// TIA Portal V17 export
// export: Created 2024-09-02T12:50:08.3817091Z, ExportSetting WithDefaults, DisplayName Totally Integrated Automation Portal, DisplayVersion V17, DisplayName TIA Portal Openness, DisplayVersion V17, DisplayName TIA Portal Version Control Interface, DisplayVersion V17, DisplayName STEP 7 Professional, DisplayVersion V17, DisplayName STEP 7 Safety, DisplayVersion V17, DisplayName WinCC Professional, DisplayVersion V17
FUNCTION_BLOCK "GraFB1_FG02_Transport_OP70"   // FB1381, GRAPH
VERSION : 0.1
// stored: AcknowledgeErrorsRequired false, AutoNumber false, GraphVersion 4.0, InitialValuesAcquisition true, IsIECCheckEnabled false, LanguageInNetworks LAD, LockOperatingMode false, PermanentILProcessingInMANMode true, SetENOAutomatically false, SkipSteps false, UDAEnableTagReadback false, WithAlarmHandling true
   // inherited from GRAPH_BASE
   VAR
      OFF_SQ_BASE : Bool;
   END_VAR
   VAR_INPUT
      OFF_SQ { ExternalWritable := 'False'} : Bool := false;   // Kette ausschalten
      INIT_SQ { ExternalWritable := 'False'} : Bool := false;   // Kette in Initialzustand versetzen
      ACK_EF { ExternalWritable := 'False'} : Bool := false;   // Alle Fehler und Störungen quittieren
      S_PREV { ExternalWritable := 'False'} : Bool := false;   // Vorherigen Schritt am Parameter S_NO ausgeben
      S_NEXT { ExternalWritable := 'False'} : Bool := false;   // Nächsten Schritt am Parameter S_NO anzeigen
      SW_AUTO { ExternalWritable := 'False'} : Bool := false;   // Automtischer Betrieb
      SW_TAP { ExternalWritable := 'False'} : Bool := false;   // Halbautomatisch/Weiterschalten mit Transition
      SW_TOP { ExternalWritable := 'False'} : Bool := false;   // Halbautomatisch/Ignoriere Transition
      SW_MAN { ExternalWritable := 'False'} : Bool := false;   // Handbetrieb
      S_SEL { ExternalWritable := 'False'} : Int := 0;   // Schritt auswählen, der an S_NO ausgegeben werden soll
      S_ON { ExternalWritable := 'False'} : Bool := false;   // Schritt aktivieren, der an Parameter S_NO anliegt
      S_OFF { ExternalWritable := 'False'} : Bool := false;   // Schritt deaktivieren, der an Parameter S_NO anliegt
      T_PUSH { ExternalWritable := 'False'} : Bool := false;   // Schaltfreigabe für Transition im halbautomatischen Betrieb
   END_VAR
   VAR_OUTPUT
      S_NO { ExternalWritable := 'False'} : Int := 0;   // Schrittnummer
      S_MORE { ExternalWritable := 'False'} : Bool := false;   // Weitere Schritte sind vorhanden und können in S_NO angezeigt werden.
      S_ACTIVE { ExternalWritable := 'False'} : Bool := false;   // Schritt, der an Parameter S_NO angezeigt wird, ist aktiv
      ERR_FLT { ExternalWritable := 'False'} : Bool := false;   // Sammelfehler Interlock oder Supervision
      AUTO_ON { ExternalWritable := 'False'} : Bool := false;   // Automatischer Betrieb eingeschaltet
      TAP_ON { ExternalWritable := 'False'} : Bool := false;   // Halbautomatischer Betrieb/Schritt mit Transition eingeschaltet
      TOP_ON { ExternalWritable := 'False'} : Bool := false;   // Halbautomatischer Betrieb/Ignoriere Transition eingeschaltet
      MAN_ON { ExternalWritable := 'False'} : Bool := false;   // Handbetrieb eingeschaltet
   END_VAR
   VAR
      extBlock { S7_SetPoint := 'True'} : "LTLL_ManualGraphExt";
   END_VAR
BEGIN
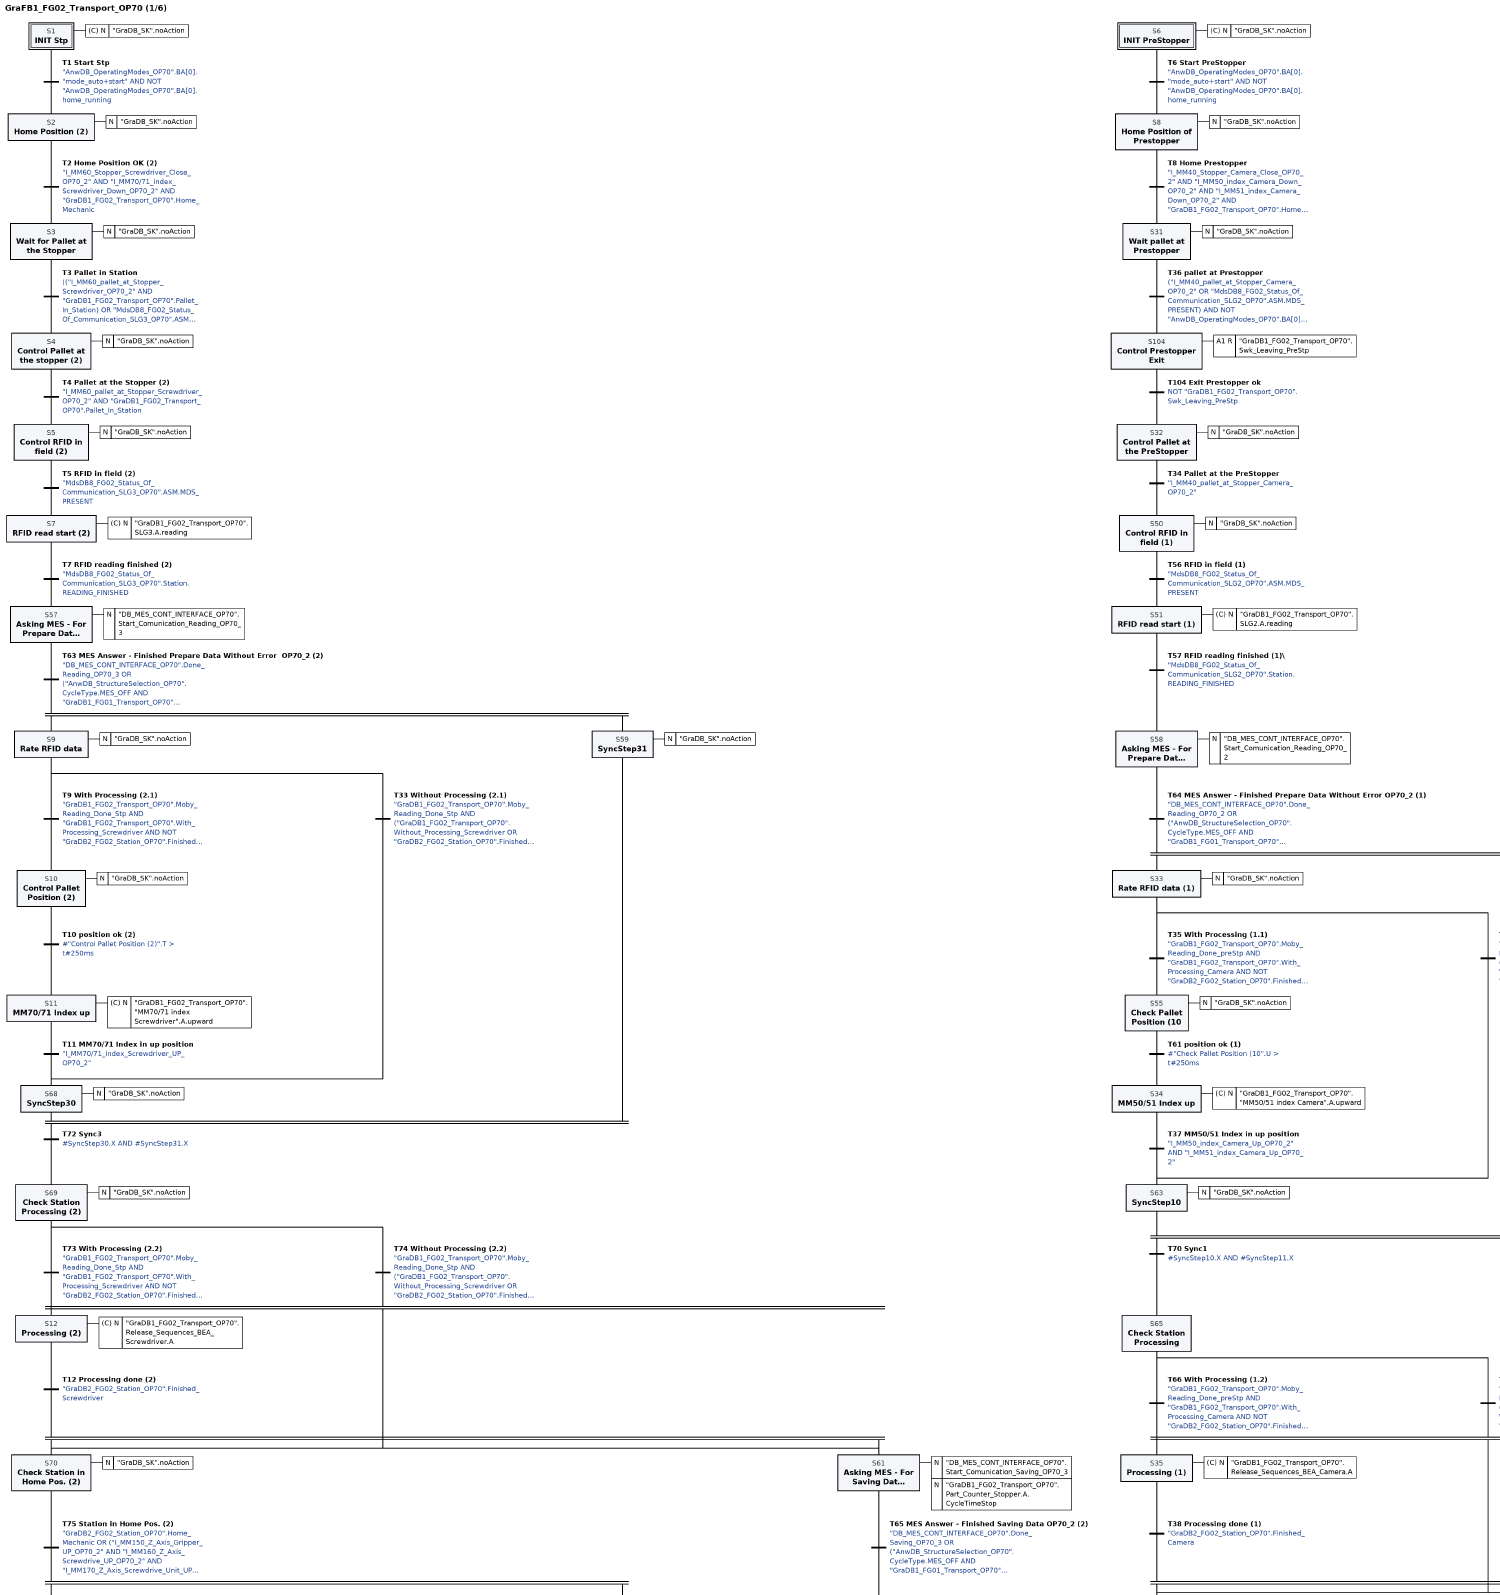
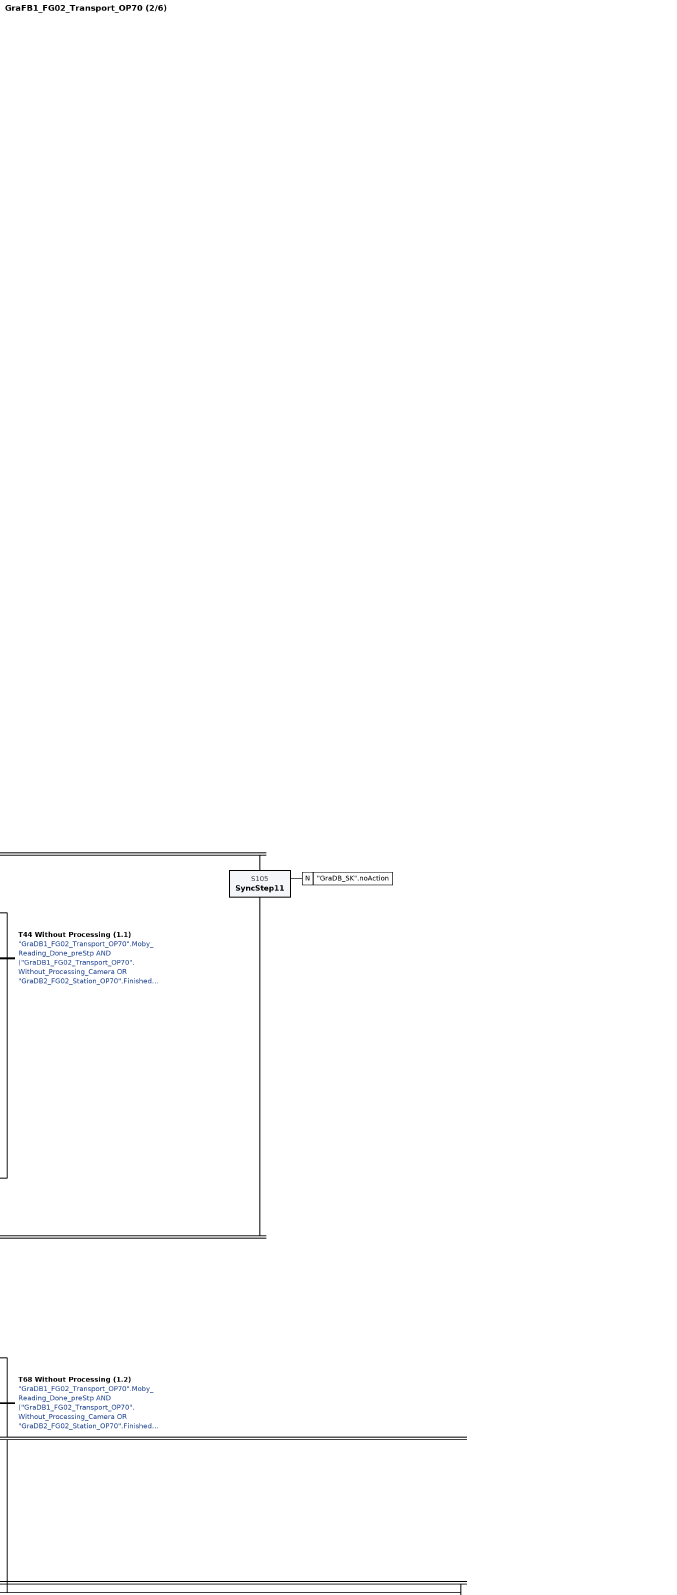
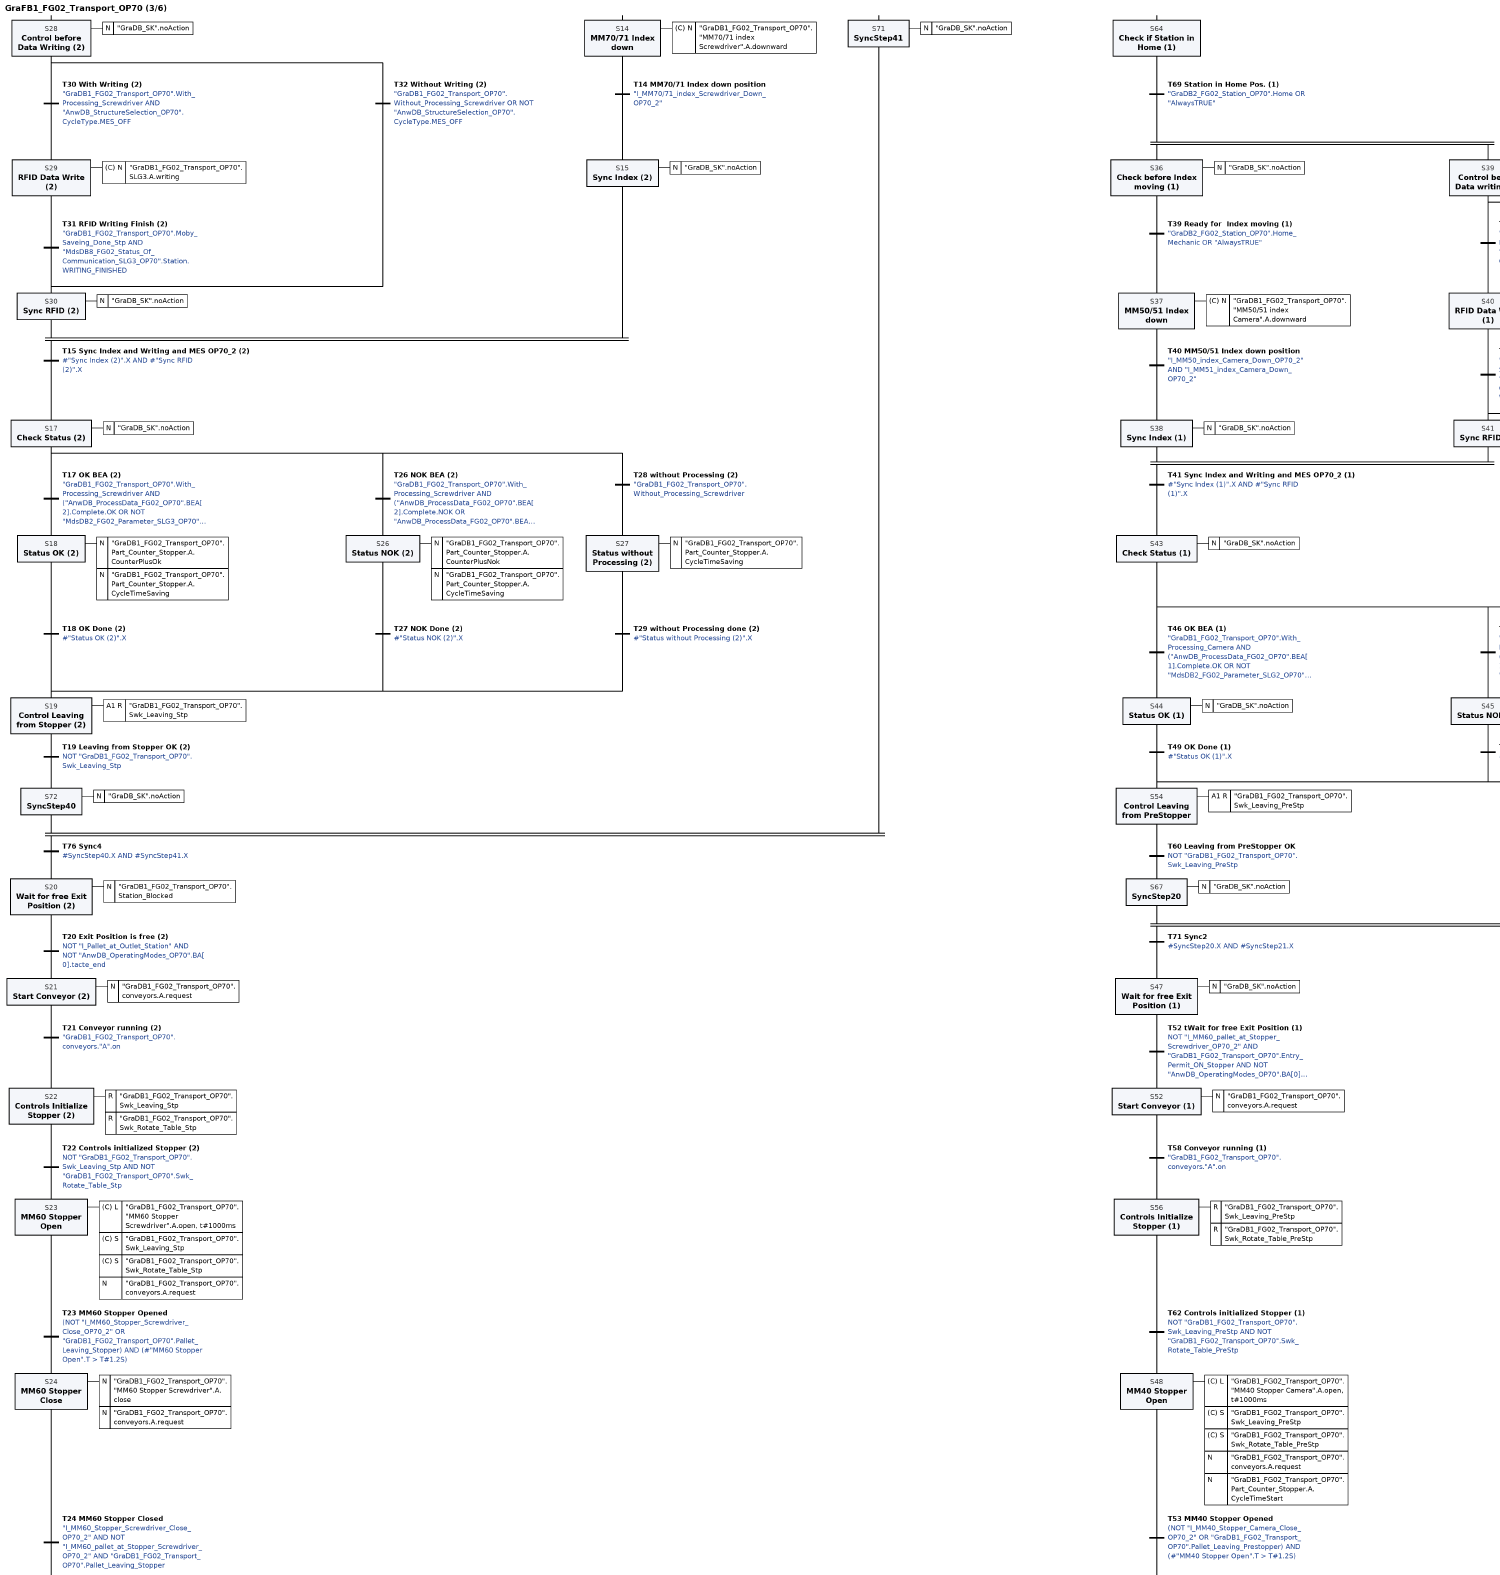
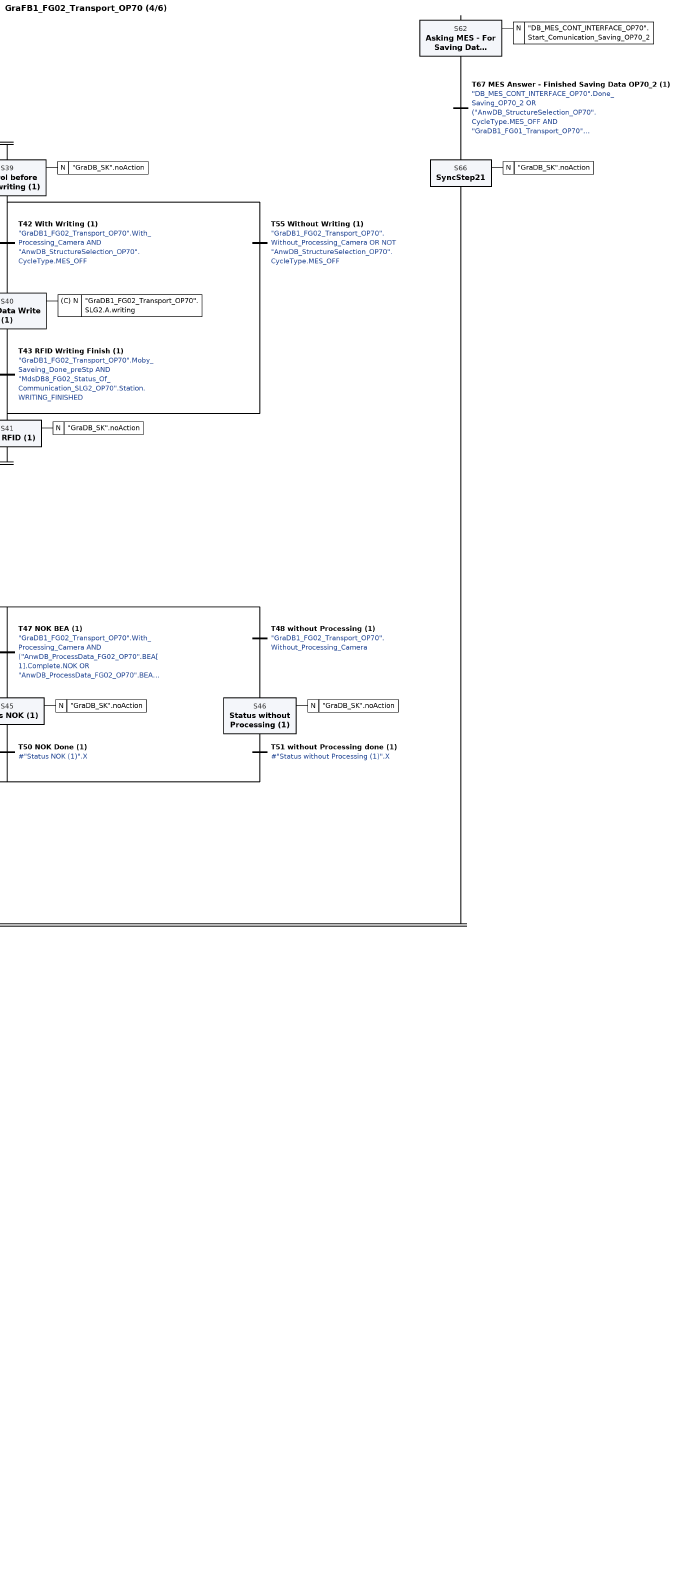
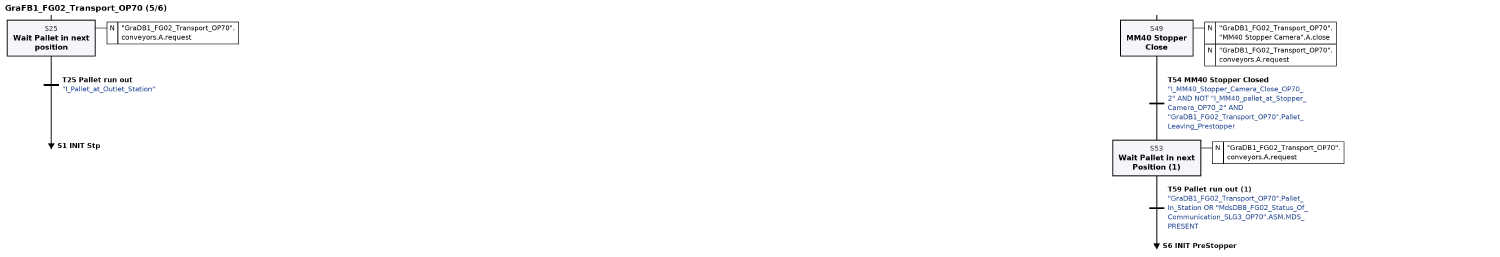
   // permanent pre-instructions
   NETWORK 1
   TITLE = HMI Lite Pass on data / HMI Lite Daten weiterreichen
      #extBlock.input := "LTLL_ManualGraphControl_OP70".screen[0].input;
   NETWORK 2
   TITLE = Instance DB Name query and pass on / Instanz DB Name abfragen und weiterreichen
      GetInstanceName(size := 0, OUT => #extBlock.input.instanceName);
   NETWORK 3
   TITLE = SK Mode
      "SysFC_SQ_Mode"(iFKT := 0, iTmsHalt := false, ioMOP := #RT_DATA.MOP);
   NETWORK 4
   TITLE = Signal change between pre-stopper and stopper / Signalwechsel Vorstopper/Stopper
      IF "GraDB1_FG02_Transport_OP70".Pallet_In_Station THEN
          "GraDB1_FG02_Transport_OP70".Swk_Leaving_PreStp := FALSE;
      END_IF;
      IF "I_Pallet_at_Outlet_Station" OR (NOT "GraDB1_FG02_Transport_OP70".Pallet_In_Station AND NOT "MdsDB8_FG02_Status_Of_Communication_SLG3_OP70".ASM.MDS_PRESENT AND NOT "I_MM60_pallet_at_Stopper_Screwdriver_OP70_2" AND "AlwaysFALSE") THEN
          "GraDB1_FG02_Transport_OP70".Swk_Leaving_Stp := FALSE;
      END_IF;
      IF "AlwaysTRUE" THEN "GraDB1_FG02_Transport_OP70".Swk_Rotate_Table_Stp := FALSE; END_IF;

   // sequencer 1: FG02 - Stopper MM60 / FG01 - Stopper
   INITIAL_STEP "INIT Stp":   // S1, max time T#10S, warning time T#7S
      interlock C := (none);   // Initialschritt / initial step
      supervision V := (none);   // Initialschritt / initial step
      (C)     N    "GraDB_SK".noAction
   END_STEP
   TRANSITION "Start Stp" FROM "INIT Stp" TO "Home Position (2)"   // T1
      := "AnwDB_OperatingModes_OP70".BA[0]."mode_auto+start" AND NOT "AnwDB_OperatingModes_OP70".BA[0].home_running;
   END_TRANSITION
   STEP "Home Position (2)":   // S2, max time T#10S, warning time T#7S
      supervision V := NOT #"Home Position OK (2)".TT AND (#"Home Position (2)".U > T#1S);
              N    "GraDB_SK".noAction
   END_STEP
   TRANSITION "Home Position OK (2)" FROM "Home Position (2)" TO "Wait for Pallet at the Stopper"   // T2
      := "I_MM60_Stopper_Screwdriver_Close_OP70_2" AND "I_MM70/71_index_Screwdriver_Down_OP70_2" AND "GraDB1_FG02_Transport_OP70".Home_Mechanic;
   END_TRANSITION
   STEP "Wait for Pallet at the Stopper":   // S3, max time T#10S, warning time T#7S
              N    "GraDB_SK".noAction
   END_STEP
   TRANSITION "Pallet in Station" FROM "Wait for Pallet at the Stopper" TO "Control Pallet at the stopper (2)"   // T3
      := (("I_MM60_pallet_at_Stopper_Screwdriver_OP70_2" AND "GraDB1_FG02_Transport_OP70".Pallet_In_Station) OR "MdsDB8_FG02_Status_Of_Communication_SLG3_OP70".ASM.MDS_PRESENT) AND NOT "AnwDB_OperatingModes_OP70".BA[0].tacte_end;
   END_TRANSITION
   STEP "Control Pallet at the stopper (2)":   // S4, max time T#10S, warning time T#7S
      supervision V := NOT #"Pallet at the Stopper (2)".TT AND (#"Control Pallet at the stopper (2)".U > T#5000mS);
              N    "GraDB_SK".noAction
   END_STEP
   TRANSITION "Pallet at the Stopper (2)" FROM "Control Pallet at the stopper (2)" TO "Control RFID in field (2)"   // T4
      := "I_MM60_pallet_at_Stopper_Screwdriver_OP70_2" AND "GraDB1_FG02_Transport_OP70".Pallet_In_Station;
   END_TRANSITION
   STEP "Rate RFID data":   // S9, max time T#10S, warning time T#7S
      interlock C := "MdsDB8_FG02_Status_Of_Communication_SLG3_OP70".Station.READING_FINISHED;
      supervision V := NOT #"With Processing (2.1)".TT AND NOT #"Without Processing (2.1)".TT AND (#"Rate RFID data".U > T#5000mS);
              N    "GraDB_SK".noAction
   END_STEP
   TRANSITION "With Processing (2.1)" FROM "Rate RFID data" TO "Control Pallet Position (2)"   // T9
      := "GraDB1_FG02_Transport_OP70".Moby_Reading_Done_Stp AND "GraDB1_FG02_Transport_OP70".With_Processing_Screwdriver AND NOT "GraDB2_FG02_Station_OP70".Finished_Screwdriver;
   END_TRANSITION
   TRANSITION "Without Processing (2.1)" FROM "Rate RFID data" TO SyncStep30   // T33
      := "GraDB1_FG02_Transport_OP70".Moby_Reading_Done_Stp AND ("GraDB1_FG02_Transport_OP70".Without_Processing_Screwdriver OR "GraDB2_FG02_Station_OP70".Finished_Screwdriver) AND (#"Rate RFID data".T > T#500MS);
   END_TRANSITION
   STEP "MM70/71 Index up":   // S11, max time T#10S, warning time T#7S
      interlock C := "I_MM150_Z_Axis_Gripper_UP_OP70_2" AND "I_MM160_Z_Axis_Screwdrive_UP_OP70_2" AND "I_MM170_Z_Axis_Screwdrive_Unit_UP_OP70_2";
      supervision V := NOT #"MM70/71 Index in up position".TT AND (#"MM70/71 Index up".U > T#5000mS);
      (C)     N    "GraDB1_FG02_Transport_OP70"."MM70/71 index Screwdriver".A.upward
   END_STEP
   TRANSITION "MM70/71 Index in up position" FROM "MM70/71 Index up" TO SyncStep30   // T11
      := "I_MM70/71_index_Screwdriver_UP_OP70_2";
   END_TRANSITION
   STEP "Processing (2)":   // S12, max time T#10S, warning time T#7S
      interlock C := "MdsDB8_FG02_Status_Of_Communication_SLG3_OP70".Station.READING_FINISHED;
      (C)     N    "GraDB1_FG02_Transport_OP70".Release_Sequences_BEA_Screwdriver.A
   END_STEP
   TRANSITION "Processing done (2)" FROM "Processing (2)" TO ("Check Station in Home Pos. (2)", "Asking MES - For Saving Data OP70_2 (2)")   // T12
      := "GraDB2_FG02_Station_OP70".Finished_Screwdriver;
   END_TRANSITION
   STEP "MM70/71 Index  down":   // S14, max time T#10S, warning time T#7S
      interlock C := "I_MM150_Z_Axis_Gripper_UP_OP70_2" AND "I_MM160_Z_Axis_Screwdrive_UP_OP70_2" AND "I_MM170_Z_Axis_Screwdrive_Unit_UP_OP70_2";
      supervision V := NOT #"MM70/71 Index down position".TT AND (#"MM70/71 Index  down".U > T#5s);
      (C)     N    "GraDB1_FG02_Transport_OP70"."MM70/71 index Screwdriver".A.downward
   END_STEP
   TRANSITION "MM70/71 Index down position" FROM "MM70/71 Index  down" TO "Sync Index (2)"   // T14
      := "I_MM70/71_index_Screwdriver_Down_OP70_2";
   END_TRANSITION
   STEP "Sync Index (2)":   // S15, max time T#10S, warning time T#7S
              N    "GraDB_SK".noAction
   END_STEP
   STEP "Control before Data Writing (2)":   // S28, max time T#10S, warning time T#7S
              N    "GraDB_SK".noAction
   END_STEP
   TRANSITION "With Writing (2)" FROM "Control before Data Writing (2)" TO "RFID Data Write (2)"   // T30
      := "GraDB1_FG02_Transport_OP70".With_Processing_Screwdriver AND "AnwDB_StructureSelection_OP70".CycleType.MES_OFF;
   END_TRANSITION
   TRANSITION "Without Writing (2)" FROM "Control before Data Writing (2)" TO "Sync RFID (2)"   // T32
      := "GraDB1_FG02_Transport_OP70".Without_Processing_Screwdriver OR NOT "AnwDB_StructureSelection_OP70".CycleType.MES_OFF;
   END_TRANSITION
   STEP "RFID Data Write (2)":   // S29, max time T#10S, warning time T#7S
      interlock C := "GraDB1_FG02_Transport_OP70".Moby_Reading_Done_Stp;
      supervision V := NOT #"RFID Writing Finish (2)".TT AND (#"RFID Data Write (2)".U > T#5000MS);
      (C)     N    "GraDB1_FG02_Transport_OP70".SLG3.A.writing
   END_STEP
   TRANSITION "RFID Writing Finish (2)" FROM "RFID Data Write (2)" TO "Sync RFID (2)"   // T31
      := "GraDB1_FG02_Transport_OP70".Moby_Saveing_Done_Stp AND "MdsDB8_FG02_Status_Of_Communication_SLG3_OP70".Station.WRITING_FINISHED;
   END_TRANSITION
   STEP "Sync RFID (2)":   // S30, max time T#10S, warning time T#7S
              N    "GraDB_SK".noAction
   END_STEP
   TRANSITION "Sync Index and Writing and MES OP70_2 (2)" FROM ("Sync Index (2)", "Sync RFID (2)") TO "Check Status (2)"   // T15
      := #"Sync Index (2)".X AND #"Sync RFID (2)".X;
   END_TRANSITION
   STEP "Check Status (2)":   // S17, max time T#10S, warning time T#7S
      supervision V := NOT #"OK BEA (2)".TT AND NOT #"OK BEA (2)".TT AND NOT #"without Processing (2)".TT AND (#"Check Status (2)".U > T#1000MS);
              N    "GraDB_SK".noAction
   END_STEP
   TRANSITION "OK BEA (2)" FROM "Check Status (2)" TO "Status OK (2)"   // T17
      := "GraDB1_FG02_Transport_OP70".With_Processing_Screwdriver AND ("AnwDB_ProcessData_FG02_OP70".BEA[2].Complete.OK OR NOT "MdsDB2_FG02_Parameter_SLG3_OP70".Release_BEA[2]) AND ("AnwDB_ProcessData_FG02_OP70".BEA[3].Complete.OK OR NOT "MdsDB2_FG02_Parameter_SLG3_OP70".Release_BEA[3]);
   END_TRANSITION
   TRANSITION "NOK BEA (2)" FROM "Check Status (2)" TO "Status NOK (2)"   // T26
      := "GraDB1_FG02_Transport_OP70".With_Processing_Screwdriver AND ("AnwDB_ProcessData_FG02_OP70".BEA[2].Complete.NOK OR "AnwDB_ProcessData_FG02_OP70".BEA[2].Complete.NOK_Active OR "AnwDB_ProcessData_FG02_OP70".BEA[3].Complete.NOK OR "AnwDB_ProcessData_FG02_OP70".BEA[3].Complete.NOK_Active);
   END_TRANSITION
   TRANSITION "without Processing (2)" FROM "Check Status (2)" TO "Status without Processing (2)"   // T28
      := "GraDB1_FG02_Transport_OP70".Without_Processing_Screwdriver;
   END_TRANSITION
   STEP "Status OK (2)":   // S18, max time T#10S, warning time T#7S
              N    "GraDB1_FG02_Transport_OP70".Part_Counter_Stopper.A.CounterPlusOk
              N    "GraDB1_FG02_Transport_OP70".Part_Counter_Stopper.A.CycleTimeSaving
   END_STEP
   TRANSITION "OK Done (2)" FROM "Status OK (2)" TO "Control Leaving from Stopper (2)"   // T18
      := #"Status OK (2)".X;
   END_TRANSITION
   STEP "Status NOK (2)":   // S26, max time T#10S, warning time T#7S
              N    "GraDB1_FG02_Transport_OP70".Part_Counter_Stopper.A.CounterPlusNok
              N    "GraDB1_FG02_Transport_OP70".Part_Counter_Stopper.A.CycleTimeSaving
   END_STEP
   TRANSITION "NOK Done (2)" FROM "Status NOK (2)" TO "Control Leaving from Stopper (2)"   // T27
      := #"Status NOK (2)".X;
   END_TRANSITION
   STEP "Status without Processing (2)":   // S27, max time T#10S, warning time T#7S
              N    "GraDB1_FG02_Transport_OP70".Part_Counter_Stopper.A.CycleTimeSaving
   END_STEP
   TRANSITION "without Processing done (2)" FROM "Status without Processing (2)" TO "Control Leaving from Stopper (2)"   // T29
      := #"Status without Processing (2)".X;
   END_TRANSITION
   STEP "Wait for free Exit Position (2)":   // S20, max time T#10S, warning time T#7S
              N    "GraDB1_FG02_Transport_OP70".Station_Blocked
   END_STEP
   TRANSITION "Exit Position is free (2)" FROM "Wait for free Exit Position (2)" TO "Start Conveyor (2)"   // T20
      := NOT "I_Pallet_at_Outlet_Station" AND NOT "AnwDB_OperatingModes_OP70".BA[0].tacte_end;
   END_TRANSITION
   STEP "MM60 Stopper Open":   // S23, max time T#10S, warning time T#7S
      interlock C := NOT "I_Pallet_at_Outlet_Station";
      supervision V := NOT #"MM60 Stopper Opened".TT AND (#"MM60 Stopper Open".U > T#5000mS);
      (C)     L    "GraDB1_FG02_Transport_OP70"."MM60 Stopper Screwdriver".A.open, t#1000ms
      (C)     S    "GraDB1_FG02_Transport_OP70".Swk_Leaving_Stp
      (C)     S    "GraDB1_FG02_Transport_OP70".Swk_Rotate_Table_Stp
              N    "GraDB1_FG02_Transport_OP70".conveyors.A.request
   END_STEP
   TRANSITION "MM60 Stopper Opened" FROM "MM60 Stopper Open" TO "MM60 Stopper Close"   // T23
      := (NOT "I_MM60_Stopper_Screwdriver_Close_OP70_2" OR "GraDB1_FG02_Transport_OP70".Pallet_Leaving_Stopper) AND (#"MM60 Stopper Open".T > T#1.2S);
   END_TRANSITION
   STEP "MM60 Stopper Close":   // S24, max time T#10S, warning time T#7S
      supervision V := NOT #"MM60 Stopper Closed".TT AND (#"MM60 Stopper Close".U > T#5000mS);
              N    "GraDB1_FG02_Transport_OP70"."MM60 Stopper Screwdriver".A.close
              N    "GraDB1_FG02_Transport_OP70".conveyors.A.request
   END_STEP
   TRANSITION "MM60 Stopper Closed" FROM "MM60 Stopper Close" TO "Wait Pallet in next position"   // T24
      := "I_MM60_Stopper_Screwdriver_Close_OP70_2" AND NOT "I_MM60_pallet_at_Stopper_Screwdriver_OP70_2" AND "GraDB1_FG02_Transport_OP70".Pallet_Leaving_Stopper;
   END_TRANSITION
   STEP "Control RFID in field (2)":   // S5, max time T#10S, warning time T#7S
      supervision V := NOT #"RFID in field (2)".TT AND (#"Control RFID in field (2)".U > T#5000mS);
              N    "GraDB_SK".noAction
   END_STEP
   TRANSITION "RFID in field (2)" FROM "Control RFID in field (2)" TO "RFID read start (2)"   // T5
      := "MdsDB8_FG02_Status_Of_Communication_SLG3_OP70".ASM.MDS_PRESENT;
   END_TRANSITION
   STEP "RFID read start (2)":   // S7, max time T#10S, warning time T#7S
      interlock C := "MdsDB8_FG02_Status_Of_Communication_SLG3_OP70".ASM.MDS_PRESENT;
      supervision V := NOT #"RFID reading finished (2)".TT AND (#"RFID read start (2)".U > T#5000mS);
      (C)     N    "GraDB1_FG02_Transport_OP70".SLG3.A.reading
   END_STEP
   TRANSITION "RFID reading finished (2)" FROM "RFID read start (2)" TO "Asking MES - For Prepare Data  OP70_2 (2)"   // T7
      := "MdsDB8_FG02_Status_Of_Communication_SLG3_OP70".Station.READING_FINISHED;
   END_TRANSITION
   STEP "Start Conveyor (2)":   // S21, max time T#10S, warning time T#7S
      supervision V := NOT #"Conveyor running (2)".TT AND (#"Start Conveyor (2)".U > T#5000MS);
              N    "GraDB1_FG02_Transport_OP70".conveyors.A.request
   END_STEP
   TRANSITION "Conveyor running (2)" FROM "Start Conveyor (2)" TO "Controls Initialize Stopper (2)"   // T21
      := "GraDB1_FG02_Transport_OP70".conveyors."A".on;
   END_TRANSITION
   STEP "Wait Pallet in next position":   // S25, max time T#10S, warning time T#7S
      supervision V := NOT #"Pallet run out".TT AND (#"Wait Pallet in next position".U > T#25000MS);
              N    "GraDB1_FG02_Transport_OP70".conveyors.A.request
   END_STEP
   TRANSITION "Pallet run out" FROM "Wait Pallet in next position" TO "INIT Stp"   // T25, jump
      := "I_Pallet_at_Outlet_Station";
   END_TRANSITION
   STEP "Control Leaving from Stopper (2)":   // S19, max time T#10S, warning time T#7S
      supervision V := NOT #"Leaving from Stopper OK (2)".TT AND (#"Control Leaving from Stopper (2)".U > T#1000MS);
          A1  R    "GraDB1_FG02_Transport_OP70".Swk_Leaving_Stp
   END_STEP
   TRANSITION "Leaving from Stopper OK (2)" FROM "Control Leaving from Stopper (2)" TO SyncStep40   // T19
      := NOT "GraDB1_FG02_Transport_OP70".Swk_Leaving_Stp;
   END_TRANSITION
   STEP "Control Pallet Position (2)":   // S10, max time T#10S, warning time T#7S
      supervision V := NOT #"position ok (2)".TT AND (#"Control Pallet Position (2)".U > T#5000MS);
              N    "GraDB_SK".noAction
   END_STEP
   TRANSITION "position ok (2)" FROM "Control Pallet Position (2)" TO "MM70/71 Index up"   // T10
      := #"Control Pallet Position (2)".T > t#250ms;
   END_TRANSITION
   STEP "Controls Initialize Stopper (2)":   // S22, max time T#10S, warning time T#7S
      supervision V := NOT #"Controls initialized Stopper (2)".TT AND (#"Controls Initialize Stopper (2)".U > T#1000MS);
              R    "GraDB1_FG02_Transport_OP70".Swk_Leaving_Stp
              R    "GraDB1_FG02_Transport_OP70".Swk_Rotate_Table_Stp
   END_STEP
   TRANSITION "Controls initialized Stopper (2)" FROM "Controls Initialize Stopper (2)" TO "MM60 Stopper Open"   // T22
      := NOT "GraDB1_FG02_Transport_OP70".Swk_Leaving_Stp AND NOT "GraDB1_FG02_Transport_OP70".Swk_Rotate_Table_Stp;
   END_TRANSITION
   STEP SyncStep30:   // S68, max time T#10S, warning time T#7S
              N    "GraDB_SK".noAction
   END_STEP
   STEP SyncStep40:   // S72, max time T#10S, warning time T#7S
              N    "GraDB_SK".noAction
   END_STEP
   STEP SyncStep31:   // S59, max time T#10S, warning time T#7S
              N    "GraDB_SK".noAction
   END_STEP
   TRANSITION Sync3 FROM (SyncStep30, SyncStep31) TO "Check Station Processing (2)"   // T72
      := #SyncStep30.X AND #SyncStep31.X;
   END_TRANSITION
   STEP "Check Station Processing (2)":   // S69, max time T#10S, warning time T#7S
              N    "GraDB_SK".noAction
   END_STEP
   TRANSITION "With Processing (2.2)" FROM "Check Station Processing (2)" TO "Processing (2)"   // T73
      := "GraDB1_FG02_Transport_OP70".Moby_Reading_Done_Stp AND "GraDB1_FG02_Transport_OP70".With_Processing_Screwdriver AND NOT "GraDB2_FG02_Station_OP70".Finished_Screwdriver;
   END_TRANSITION
   TRANSITION "Without Processing (2.2)" FROM "Check Station Processing (2)" TO ("Check Station in Home Pos. (2)", "Asking MES - For Saving Data OP70_2 (2)")   // T74
      := "GraDB1_FG02_Transport_OP70".Moby_Reading_Done_Stp AND ("GraDB1_FG02_Transport_OP70".Without_Processing_Screwdriver OR "GraDB2_FG02_Station_OP70".Finished_Screwdriver) AND (#"Check Station Processing (2)".T > t#500ms);
   END_TRANSITION
   STEP "Check Station in Home Pos. (2)":   // S70, max time T#10S, warning time T#7S
      supervision V := NOT #"Station in Home Pos. (2)".TT AND (#"Check Station in Home Pos. (2)".U > T#5s);
              N    "GraDB_SK".noAction
   END_STEP
   TRANSITION "Station in Home Pos. (2)" FROM "Check Station in Home Pos. (2)" TO ("Control before Data Writing (2)", "MM70/71 Index  down")   // T75
      := "GraDB2_FG02_Station_OP70".Home_Mechanic OR ("I_MM150_Z_Axis_Gripper_UP_OP70_2" AND "I_MM160_Z_Axis_Screwdrive_UP_OP70_2" AND "I_MM170_Z_Axis_Screwdrive_Unit_UP_OP70_2");
   END_TRANSITION
   STEP SyncStep41:   // S71, max time T#10S, warning time T#7S
              N    "GraDB_SK".noAction
   END_STEP
   TRANSITION Sync4 FROM (SyncStep40, SyncStep41) TO "Wait for free Exit Position (2)"   // T76
      := #SyncStep40.X AND #SyncStep41.X;
   END_TRANSITION
   STEP "Asking MES - For Saving Data OP70_2 (2)":   // S61, max time T#10S, warning time T#7S
      interlock C := "MdsDB8_FG02_Status_Of_Communication_SLG3_OP70".ASM.MDS_PRESENT;
      supervision V := NOT #"MES Answer - Finished Saving Data OP70_2 (2)".TT AND (#"Asking MES - For Saving Data OP70_2 (2)".U > T#5000mS) AND "AlwaysFALSE";
              N    "DB_MES_CONT_INTERFACE_OP70".Start_Comunication_Saving_OP70_3
              N    "GraDB1_FG02_Transport_OP70".Part_Counter_Stopper.A.CycleTimeStop
   END_STEP
   TRANSITION "MES Answer - Finished Saving Data OP70_2 (2)" FROM "Asking MES - For Saving Data OP70_2 (2)" TO SyncStep41   // T65
      := "DB_MES_CONT_INTERFACE_OP70".Done_Saving_OP70_3 OR ("AnwDB_StructureSelection_OP70".CycleType.MES_OFF AND "GraDB1_FG01_Transport_OP70".Tracebility_off) OR "AnwDB_StructureSelection_OP70".UserDefine.IbmMode;
   END_TRANSITION
   STEP "Asking MES - For Prepare Data  OP70_2 (2)":   // S57, max time T#10S, warning time T#7S
      interlock C := "MdsDB8_FG02_Status_Of_Communication_SLG3_OP70".ASM.MDS_PRESENT;
      supervision V := NOT #"MES Answer - Finished Prepare Data Without Error  OP70_2 (2)".TT AND (#"Asking MES - For Prepare Data  OP70_2 (2)".U > T#7s);
              N    "DB_MES_CONT_INTERFACE_OP70".Start_Comunication_Reading_OP70_3
   END_STEP
   TRANSITION "MES Answer - Finished Prepare Data Without Error  OP70_2 (2)" FROM "Asking MES - For Prepare Data  OP70_2 (2)" TO ("Rate RFID data", SyncStep31)   // T63
      := "DB_MES_CONT_INTERFACE_OP70".Done_Reading_OP70_3 OR ("AnwDB_StructureSelection_OP70".CycleType.MES_OFF AND "GraDB1_FG01_Transport_OP70".Tracebility_off) OR "AnwDB_StructureSelection_OP70".UserDefine.IbmMode;
   END_TRANSITION

   // sequencer 2: FG02 - PreStopper MM40 / FG01 - Vorstopper
   INITIAL_STEP "INIT PreStopper":   // S6, max time T#10S, warning time T#7S
      interlock C := (none);   // Initialschritt / initial step
      supervision V := (none);   // Initialschritt / initial step
      (C)     N    "GraDB_SK".noAction
   END_STEP
   TRANSITION "Start PreStopper" FROM "INIT PreStopper" TO "Home Position of Prestopper"   // T6
      := "AnwDB_OperatingModes_OP70".BA[0]."mode_auto+start" AND NOT "AnwDB_OperatingModes_OP70".BA[0].home_running;
   END_TRANSITION
   STEP "Home Position of Prestopper":   // S8, max time T#10S, warning time T#7S
      supervision V := NOT #"Home Prestopper".TT AND (#"Home Position of Prestopper".U > T#1S);
              N    "GraDB_SK".noAction
   END_STEP
   TRANSITION "Home Prestopper" FROM "Home Position of Prestopper" TO "Wait pallet at Prestopper"   // T8
      := "I_MM40_Stopper_Camera_Close_OP70_2" AND "I_MM50_index_Camera_Down_OP70_2" AND "I_MM51_index_Camera_Down_OP70_2" AND "GraDB1_FG02_Transport_OP70".Home_Mechanic;
   END_TRANSITION
   STEP "Sync Index (1)":   // S38, max time T#10S, warning time T#7S
              N    "GraDB_SK".noAction
   END_STEP
   STEP "Control before Data writing (1)":   // S39, max time T#10S, warning time T#7S
              N    "GraDB_SK".noAction
   END_STEP
   TRANSITION "With Writing (1)" FROM "Control before Data writing (1)" TO "RFID Data Write (1)"   // T42
      := "GraDB1_FG02_Transport_OP70".With_Processing_Camera AND "AnwDB_StructureSelection_OP70".CycleType.MES_OFF;
   END_TRANSITION
   TRANSITION "Without Writing (1)" FROM "Control before Data writing (1)" TO "Sync RFID (1)"   // T55
      := "GraDB1_FG02_Transport_OP70".Without_Processing_Camera OR NOT "AnwDB_StructureSelection_OP70".CycleType.MES_OFF;
   END_TRANSITION
   STEP "Rate RFID data (1)":   // S33, max time T#10S, warning time T#7S
      interlock C := "AlwaysTRUE";
      supervision V := NOT #"With Processing (1.1)".TT AND NOT #"Without Processing (1.1)".TT AND (#"Rate RFID data (1)".U > T#5000mS);
              N    "GraDB_SK".noAction
   END_STEP
   TRANSITION "With Processing (1.1)" FROM "Rate RFID data (1)" TO "Check Pallet Position (10"   // T35
      := "GraDB1_FG02_Transport_OP70".Moby_Reading_Done_preStp AND "GraDB1_FG02_Transport_OP70".With_Processing_Camera AND NOT "GraDB2_FG02_Station_OP70".Finished_Camera;
   END_TRANSITION
   TRANSITION "Without Processing (1.1)" FROM "Rate RFID data (1)" TO SyncStep10   // T44
      := "GraDB1_FG02_Transport_OP70".Moby_Reading_Done_preStp AND ("GraDB1_FG02_Transport_OP70".Without_Processing_Camera OR "GraDB2_FG02_Station_OP70".Finished_Camera) AND (#"Rate RFID data (1)".T > T#500MS);
   END_TRANSITION
   STEP "Processing (1)":   // S35, max time T#10S, warning time T#7S
      interlock C := "I_MM50_index_Camera_Up_OP70_2" AND "I_MM51_index_Camera_Up_OP70_2" AND "MdsDB8_FG02_Status_Of_Communication_SLG2_OP70".Station.READING_FINISHED;
      (C)     N    "GraDB1_FG02_Transport_OP70".Release_Sequences_BEA_Camera.A
   END_STEP
   TRANSITION "Processing done (1)" FROM "Processing (1)" TO ("Check if Station in Home (1)", "Asking MES - For Saving Data OP70_2 (1)")   // T38
      := "GraDB2_FG02_Station_OP70".Finished_Camera;
   END_TRANSITION
   STEP "RFID Data Write (1)":   // S40, max time T#10S, warning time T#7S
      interlock C := "GraDB1_FG02_Transport_OP70".Moby_Reading_Done_preStp;
      supervision V := NOT #"RFID Writing Finish (1)".TT AND (#"RFID Data Write (1)".U > T#5000MS);
      (C)     N    "GraDB1_FG02_Transport_OP70".SLG2.A.writing
   END_STEP
   TRANSITION "RFID Writing Finish (1)" FROM "RFID Data Write (1)" TO "Sync RFID (1)"   // T43
      := "GraDB1_FG02_Transport_OP70".Moby_Saveing_Done_preStp AND "MdsDB8_FG02_Status_Of_Communication_SLG2_OP70".Station.WRITING_FINISHED;
   END_TRANSITION
   STEP "Check before Index moving (1)":   // S36, max time T#10S, warning time T#7S
      interlock C := "AlwaysTRUE";
      supervision V := NOT #"Ready for  Index moving (1)".TT AND (#"Check before Index moving (1)".U > T#5000MS);
              N    "GraDB_SK".noAction
   END_STEP
   TRANSITION "Ready for  Index moving (1)" FROM "Check before Index moving (1)" TO "MM50/51 Index  down"   // T39
      := "GraDB2_FG02_Station_OP70".Home_Mechanic OR "AlwaysTRUE";
   END_TRANSITION
   STEP "MM50/51 Index up":   // S34, max time T#10S, warning time T#7S
      supervision V := NOT #"MM50/51 Index in up position".TT AND (#"MM50/51 Index up".U > T#5000mS);
      (C)     N    "GraDB1_FG02_Transport_OP70"."MM50/51 index Camera".A.upward
   END_STEP
   TRANSITION "MM50/51 Index in up position" FROM "MM50/51 Index up" TO SyncStep10   // T37
      := "I_MM50_index_Camera_Up_OP70_2" AND "I_MM51_index_Camera_Up_OP70_2";
   END_TRANSITION
   STEP "MM50/51 Index  down":   // S37, max time T#10S, warning time T#7S
      interlock C := "AlwaysTRUE";
      supervision V := NOT #"MM50/51 Index down position".TT AND (#"MM50/51 Index  down".U > T#5000mS);
      (C)     N    "GraDB1_FG02_Transport_OP70"."MM50/51 index Camera".A.downward
   END_STEP
   TRANSITION "MM50/51 Index down position" FROM "MM50/51 Index  down" TO "Sync Index (1)"   // T40
      := "I_MM50_index_Camera_Down_OP70_2" AND "I_MM51_index_Camera_Down_OP70_2";
   END_TRANSITION
   STEP "Wait pallet at Prestopper":   // S31, max time T#10S, warning time T#7S
              N    "GraDB_SK".noAction
   END_STEP
   TRANSITION "pallet at Prestopper" FROM "Wait pallet at Prestopper" TO "Control Prestopper Exit"   // T36
      := ("I_MM40_pallet_at_Stopper_Camera_OP70_2" OR "MdsDB8_FG02_Status_Of_Communication_SLG2_OP70".ASM.MDS_PRESENT) AND NOT "AnwDB_OperatingModes_OP70".BA[0].tacte_end;
   END_TRANSITION
   STEP "Control Pallet at the PreStopper":   // S32, max time T#10S, warning time T#7S
      supervision V := NOT #"Pallet at the PreStopper".TT AND (#"Control Pallet at the PreStopper".U > T#5000mS);
              N    "GraDB_SK".noAction
   END_STEP
   TRANSITION "Pallet at the PreStopper" FROM "Control Pallet at the PreStopper" TO "Control RFID in field (1)"   // T34
      := "I_MM40_pallet_at_Stopper_Camera_OP70_2";
   END_TRANSITION
   STEP "Sync RFID (1)":   // S41, max time T#10S, warning time T#7S
              N    "GraDB_SK".noAction
   END_STEP
   TRANSITION "Sync Index and Writing and MES OP70_2 (1)" FROM ("Sync Index (1)", "Sync RFID (1)") TO "Check Status (1)"   // T41
      := #"Sync Index (1)".X AND #"Sync RFID (1)".X;
   END_TRANSITION
   STEP "Check Status (1)":   // S43, max time T#10S, warning time T#7S
      supervision V := NOT #"OK BEA (1)".TT AND NOT #"OK BEA (1)".TT AND NOT #"without Processing (1)".TT AND (#"Check Status (1)".U > T#1000MS);
              N    "GraDB_SK".noAction
   END_STEP
   TRANSITION "OK BEA (1)" FROM "Check Status (1)" TO "Status OK (1)"   // T46
      := "GraDB1_FG02_Transport_OP70".With_Processing_Camera AND ("AnwDB_ProcessData_FG02_OP70".BEA[1].Complete.OK OR NOT "MdsDB2_FG02_Parameter_SLG2_OP70".Release_BEA[1]);
   END_TRANSITION
   TRANSITION "NOK BEA (1)" FROM "Check Status (1)" TO "Status NOK (1)"   // T47
      := "GraDB1_FG02_Transport_OP70".With_Processing_Camera AND ("AnwDB_ProcessData_FG02_OP70".BEA[1].Complete.NOK OR "AnwDB_ProcessData_FG02_OP70".BEA[1].Complete.NOK_Active);
   END_TRANSITION
   TRANSITION "without Processing (1)" FROM "Check Status (1)" TO "Status without Processing (1)"   // T48
      := "GraDB1_FG02_Transport_OP70".Without_Processing_Camera;
   END_TRANSITION
   STEP "Status OK (1)":   // S44, max time T#10S, warning time T#7S
              N    "GraDB_SK".noAction
   END_STEP
   TRANSITION "OK Done (1)" FROM "Status OK (1)" TO "Control Leaving from PreStopper"   // T49
      := #"Status OK (1)".X;
   END_TRANSITION
   STEP "Status NOK (1)":   // S45, max time T#10S, warning time T#7S
              N    "GraDB_SK".noAction
   END_STEP
   TRANSITION "NOK Done (1)" FROM "Status NOK (1)" TO "Control Leaving from PreStopper"   // T50
      := #"Status NOK (1)".X;
   END_TRANSITION
   STEP "Status without Processing (1)":   // S46, max time T#10S, warning time T#7S
              N    "GraDB_SK".noAction
   END_STEP
   TRANSITION "without Processing done (1)" FROM "Status without Processing (1)" TO "Control Leaving from PreStopper"   // T51
      := #"Status without Processing (1)".X;
   END_TRANSITION
   STEP "Wait for free Exit Position (1)":   // S47, max time T#10S, warning time T#7S
              N    "GraDB_SK".noAction
   END_STEP
   TRANSITION "tWait for free Exit Position (1)" FROM "Wait for free Exit Position (1)" TO "Start Conveyor (1)"   // T52
      := NOT "I_MM60_pallet_at_Stopper_Screwdriver_OP70_2" AND "GraDB1_FG02_Transport_OP70".Entry_Permit_ON_Stopper AND NOT "AnwDB_OperatingModes_OP70".BA[0].tacte_end;
   END_TRANSITION
   STEP "MM40 Stopper Open":   // S48, max time T#10S, warning time T#7S
      interlock C := "I_MM50_index_Camera_Down_OP70_2" AND "I_MM51_index_Camera_Down_OP70_2" AND NOT "I_MM60_pallet_at_Stopper_Screwdriver_OP70_2" AND "I_MM70/71_index_Screwdriver_Down_OP70_2" AND "I_MM150_Z_Axis_Gripper_UP_OP70_2" AND "I_MM160_Z_Axis_Screwdrive_UP_OP70_2" AND "I_MM170_Z_Axis_Screwdrive_Unit_UP_OP70_2";
      supervision V := NOT #"MM40 Stopper Opened".TT AND (#"MM40 Stopper Open".U > T#5000mS);
      (C)     L    "GraDB1_FG02_Transport_OP70"."MM40 Stopper Camera".A.open, t#1000ms
      (C)     S    "GraDB1_FG02_Transport_OP70".Swk_Leaving_PreStp
      (C)     S    "GraDB1_FG02_Transport_OP70".Swk_Rotate_Table_PreStp
              N    "GraDB1_FG02_Transport_OP70".conveyors.A.request
              N    "GraDB1_FG02_Transport_OP70".Part_Counter_Stopper.A.CycleTimeStart
   END_STEP
   TRANSITION "MM40 Stopper Opened" FROM "MM40 Stopper Open" TO "MM40 Stopper Close"   // T53
      := (NOT "I_MM40_Stopper_Camera_Close_OP70_2" OR "GraDB1_FG02_Transport_OP70".Pallet_Leaving_Prestopper) AND (#"MM40 Stopper Open".T > T#1.2S);
   END_TRANSITION
   STEP "MM40 Stopper Close":   // S49, max time T#10S, warning time T#7S
      supervision V := NOT #"MM40 Stopper Closed".TT AND (#"MM40 Stopper Close".U > T#5000mS);
              N    "GraDB1_FG02_Transport_OP70"."MM40 Stopper Camera".A.close
              N    "GraDB1_FG02_Transport_OP70".conveyors.A.request
   END_STEP
   TRANSITION "MM40 Stopper Closed" FROM "MM40 Stopper Close" TO "Wait Pallet in next Position (1)"   // T54
      := "I_MM40_Stopper_Camera_Close_OP70_2" AND NOT "I_MM40_pallet_at_Stopper_Camera_OP70_2" AND "GraDB1_FG02_Transport_OP70".Pallet_Leaving_Prestopper;
   END_TRANSITION
   STEP "Control RFID in field (1)":   // S50, max time T#10S, warning time T#7S
      supervision V := NOT #"RFID in field (1)".TT AND (#"Control RFID in field (1)".U > T#5000mS);
              N    "GraDB_SK".noAction
   END_STEP
   TRANSITION "RFID in field (1)" FROM "Control RFID in field (1)" TO "RFID read start (1)"   // T56
      := "MdsDB8_FG02_Status_Of_Communication_SLG2_OP70".ASM.MDS_PRESENT;
   END_TRANSITION
   STEP "RFID read start (1)":   // S51, max time T#10S, warning time T#7S
      interlock C := "MdsDB8_FG02_Status_Of_Communication_SLG2_OP70".ASM.MDS_PRESENT;
      supervision V := NOT #"RFID reading finished (1)\".TT AND (#"RFID read start (1)".U > T#5000mS);
      (C)     N    "GraDB1_FG02_Transport_OP70".SLG2.A.reading
   END_STEP
   TRANSITION "RFID reading finished (1)\" FROM "RFID read start (1)" TO "Asking MES - For Prepare Data OP70_2 (1)"   // T57
      := "MdsDB8_FG02_Status_Of_Communication_SLG2_OP70".Station.READING_FINISHED;
   END_TRANSITION
   STEP "Start Conveyor (1)":   // S52, max time T#10S, warning time T#7S
      supervision V := NOT #"Conveyor running (1)".TT AND (#"Start Conveyor (1)".U > T#5000MS);
              N    "GraDB1_FG02_Transport_OP70".conveyors.A.request
   END_STEP
   TRANSITION "Conveyor running (1)" FROM "Start Conveyor (1)" TO "Controls Initialize Stopper (1)"   // T58
      := "GraDB1_FG02_Transport_OP70".conveyors."A".on;
   END_TRANSITION
   STEP "Wait Pallet in next Position (1)":   // S53, max time T#10S, warning time T#7S
      supervision V := NOT #"Pallet run out (1)".TT AND (#"Wait Pallet in next Position (1)".U > T#15000MS);
              N    "GraDB1_FG02_Transport_OP70".conveyors.A.request
   END_STEP
   TRANSITION "Pallet run out (1)" FROM "Wait Pallet in next Position (1)" TO "INIT PreStopper"   // T59, jump
      := "GraDB1_FG02_Transport_OP70".Pallet_In_Station OR "MdsDB8_FG02_Status_Of_Communication_SLG3_OP70".ASM.MDS_PRESENT;
   END_TRANSITION
   STEP "Control Leaving from PreStopper":   // S54, max time T#10S, warning time T#7S
      supervision V := NOT #"Leaving from PreStopper OK".TT AND (#"Control Leaving from PreStopper".U > T#1000MS);
          A1  R    "GraDB1_FG02_Transport_OP70".Swk_Leaving_PreStp
   END_STEP
   TRANSITION "Leaving from PreStopper OK" FROM "Control Leaving from PreStopper" TO SyncStep20   // T60
      := NOT "GraDB1_FG02_Transport_OP70".Swk_Leaving_PreStp;
   END_TRANSITION
   STEP "Check Pallet Position (10":   // S55, max time T#10S, warning time T#7S
      supervision V := NOT #"position ok (1)".TT AND (#"Check Pallet Position (10".U > T#5000MS);
              N    "GraDB_SK".noAction
   END_STEP
   TRANSITION "position ok (1)" FROM "Check Pallet Position (10" TO "MM50/51 Index up"   // T61
      := #"Check Pallet Position (10".U > t#250ms;
   END_TRANSITION
   STEP "Controls Initialize Stopper (1)":   // S56, max time T#10S, warning time T#7S
      supervision V := NOT #"Controls initialized Stopper (1)".TT AND (#"Controls Initialize Stopper (1)".U > T#1000MS);
              R    "GraDB1_FG02_Transport_OP70".Swk_Leaving_PreStp
              R    "GraDB1_FG02_Transport_OP70".Swk_Rotate_Table_PreStp
   END_STEP
   TRANSITION "Controls initialized Stopper (1)" FROM "Controls Initialize Stopper (1)" TO "MM40 Stopper Open"   // T62
      := NOT "GraDB1_FG02_Transport_OP70".Swk_Leaving_PreStp AND NOT "GraDB1_FG02_Transport_OP70".Swk_Rotate_Table_PreStp;
   END_TRANSITION
   STEP SyncStep10:   // S63, max time T#10S, warning time T#7S
              N    "GraDB_SK".noAction
   END_STEP
   STEP "Control Prestopper Exit":   // S104, max time T#10S, warning time T#7S
      supervision V := NOT #"Exit Prestopper ok".TT AND (#"Control Prestopper Exit".U > T#1000MS);
          A1  R    "GraDB1_FG02_Transport_OP70".Swk_Leaving_PreStp
   END_STEP
   TRANSITION "Exit Prestopper ok" FROM "Control Prestopper Exit" TO "Control Pallet at the PreStopper"   // T104
      := NOT "GraDB1_FG02_Transport_OP70".Swk_Leaving_PreStp;
   END_TRANSITION
   STEP SyncStep11:   // S105, max time T#10S, warning time T#7S
              N    "GraDB_SK".noAction
   END_STEP
   TRANSITION Sync1 FROM (SyncStep10, SyncStep11) TO "Check Station Processing"   // T70
      := #SyncStep10.X AND #SyncStep11.X;
   END_TRANSITION
   STEP "Check if Station in Home (1)":   // S64, max time T#10S, warning time T#7S
   END_STEP
   TRANSITION "Station in Home Pos. (1)" FROM "Check if Station in Home (1)" TO ("Check before Index moving (1)", "Control before Data writing (1)")   // T69
      := "GraDB2_FG02_Station_OP70".Home OR "AlwaysTRUE";
   END_TRANSITION
   STEP "Check Station Processing":   // S65, max time T#10S, warning time T#7S
   END_STEP
   TRANSITION "With Processing (1.2)" FROM "Check Station Processing" TO "Processing (1)"   // T66
      := "GraDB1_FG02_Transport_OP70".Moby_Reading_Done_preStp AND "GraDB1_FG02_Transport_OP70".With_Processing_Camera AND NOT "GraDB2_FG02_Station_OP70".Finished_Camera;
   END_TRANSITION
   TRANSITION "Without Processing (1.2)" FROM "Check Station Processing" TO ("Check if Station in Home (1)", "Asking MES - For Saving Data OP70_2 (1)")   // T68
      := "GraDB1_FG02_Transport_OP70".Moby_Reading_Done_preStp AND ("GraDB1_FG02_Transport_OP70".Without_Processing_Camera OR "GraDB2_FG02_Station_OP70".Finished_Camera) AND (#"Check Station Processing".T > t#500ms);
   END_TRANSITION
   STEP SyncStep20:   // S67, max time T#10S, warning time T#7S
              N    "GraDB_SK".noAction
   END_STEP
   STEP SyncStep21:   // S66, max time T#10S, warning time T#7S
              N    "GraDB_SK".noAction
   END_STEP
   TRANSITION Sync2 FROM (SyncStep20, SyncStep21) TO "Wait for free Exit Position (1)"   // T71
      := #SyncStep20.X AND #SyncStep21.X;
   END_TRANSITION
   STEP "Asking MES - For Saving Data OP70_2 (1)":   // S62, max time T#10S, warning time T#7S
      interlock C := "MdsDB8_FG02_Status_Of_Communication_SLG2_OP70".ASM.MDS_PRESENT;
      supervision V := NOT #"MES Answer - Finished Saving Data OP70_2 (1)".TT AND (#"Asking MES - For Saving Data OP70_2 (1)".U > T#5000mS) AND "AlwaysFALSE";
              N    "DB_MES_CONT_INTERFACE_OP70".Start_Comunication_Saving_OP70_2
   END_STEP
   TRANSITION "MES Answer - Finished Saving Data OP70_2 (1)" FROM "Asking MES - For Saving Data OP70_2 (1)" TO SyncStep21   // T67
      := "DB_MES_CONT_INTERFACE_OP70".Done_Saving_OP70_2 OR ("AnwDB_StructureSelection_OP70".CycleType.MES_OFF AND "GraDB1_FG01_Transport_OP70".Tracebility_off) OR "AnwDB_StructureSelection_OP70".UserDefine.IbmMode;
   END_TRANSITION
   STEP "Asking MES - For Prepare Data OP70_2 (1)":   // S58, max time T#10S, warning time T#7S
      interlock C := "MdsDB8_FG02_Status_Of_Communication_SLG2_OP70".ASM.MDS_PRESENT;
      supervision V := NOT #"MES Answer - Finished Prepare Data Without Error OP70_2 (1)".TT AND (#"Asking MES - For Prepare Data OP70_2 (1)".U > T#7s);
              N    "DB_MES_CONT_INTERFACE_OP70".Start_Comunication_Reading_OP70_2
   END_STEP
   TRANSITION "MES Answer - Finished Prepare Data Without Error OP70_2 (1)" FROM "Asking MES - For Prepare Data OP70_2 (1)" TO ("Rate RFID data (1)", SyncStep11)   // T64
      := "DB_MES_CONT_INTERFACE_OP70".Done_Reading_OP70_2 OR ("AnwDB_StructureSelection_OP70".CycleType.MES_OFF AND "GraDB1_FG01_Transport_OP70".Tracebility_off) OR "AnwDB_StructureSelection_OP70".UserDefine.IbmMode;
   END_TRANSITION

   // permanent post-instructions
   NETWORK 1
   TITLE = Move interlocks from Ext block to ManualGraphControl DB / Interlocks vom Ext-Block zum ManualGraphControl DB rangieren
      "LTLL_ManualGraphInterlock"(ManualGraphExtOutput := #extBlock.output,
                              ManualGraphControlScreen := "LTLL_ManualGraphControl_OP70".screen[0]);
   NETWORK 2
   TITLE = Report step error / Schrittkettenfehler melden
      "SysFC_NumOfSQErrors"(FLT := #RT_DATA.SQ_FLAGS.ERR_FLT,
                            Fault_SQ := "AnwDB_OperatingModes_OP70".BA[0].error_report_SK,
                            NumOf_Fault_SQ := "AnwDB_ZP_Alarm_OP70".FaultsNoSK_ST1);
   NETWORK 3
   TITLE = Basic position Step chain / Grundstellung Schrittkette
      "GraDB1_FG02_Transport_OP70".Home_SQ := (#"INIT PreStopper".X OR #"Wait pallet at Prestopper".X OR #"Wait for free Exit Position (1)".X) AND (#"INIT Stp".X OR #"Wait for Pallet at the Stopper".X OR #"Wait for free Exit Position (2)".X);
   NETWORK 4
   TITLE = WT is run out Vorstopper / Stopper / WT ist Ausgelaufen Vorstopper / Stopper
      "GraDB1_FG02_Transport_OP70".Pallet_Leaving_Prestopper := (#"MM40 Stopper Open".X OR #"MM40 Stopper Close".X) AND ((NOT "I_MM40_pallet_at_Stopper_Camera_OP70_2" AND NOT "MdsDB8_FG02_Status_Of_Communication_SLG2_OP70".ASM.MDS_PRESENT) OR "GraDB1_FG02_Transport_OP70".Pallet_Leaving_Prestopper);
      "GraDB1_FG02_Transport_OP70".Pallet_Leaving_Stopper := (#"MM60 Stopper Open".X OR #"MM60 Stopper Close".X) AND ((NOT "I_MM60_pallet_at_Stopper_Screwdriver_OP70_2" AND NOT "MdsDB8_FG02_Status_Of_Communication_SLG3_OP70".ASM.MDS_PRESENT) OR "GraDB1_FG02_Transport_OP70".Pallet_Leaving_Stopper);
   NETWORK 5
   TITLE = Enable inlet / Freigabe Einlauf
      "GraDB1_FG02_Transport_OP70".Entry_Permit_ON_Stopper := ((NOT "MdsDB8_FG02_Status_Of_Communication_SLG3_OP70".ASM.MDS_PRESENT AND NOT "I_MM60_pallet_at_Stopper_Screwdriver_OP70_2") OR (#"MM60 Stopper Open".X AND NOT #"MM60 Stopper Open".LA AND "AlwaysFALSE") OR #"MM60 Stopper Close".X) AND "GraDB1_FG02_Transport_OP70".Home_Mechanic AND "I_MM70/71_index_Screwdriver_Down_OP70_2" AND "I_MM150_Z_Axis_Gripper_UP_OP70_2" AND "I_MM160_Z_Axis_Screwdrive_UP_OP70_2" AND "I_MM170_Z_Axis_Screwdrive_Unit_UP_OP70_2";
      "GraDB1_FG02_Transport_OP70".Entry_Permit_ON_PreStopper := ((#"Wait pallet at Prestopper".X AND NOT "MdsDB8_FG02_Status_Of_Communication_SLG2_OP70".ASM.MDS_PRESENT AND NOT "I_MM40_pallet_at_Stopper_Camera_OP70_2") OR (#"MM40 Stopper Open".X AND NOT #"MM40 Stopper Open".LA AND "AlwaysFALSE") OR #"MM40 Stopper Close".X) AND "I_MM50_index_Camera_Down_OP70_2" AND "I_MM51_index_Camera_Down_OP70_2";
   NETWORK 6
   TITLE = Wait for WT / Warte auf WT
      "GraDB1_FG02_Transport_OP70".Wait_For_Pallet := #"Wait pallet at Prestopper".X AND #"Wait for Pallet at the Stopper".X;
END_FUNCTION_BLOCK
